Yaskawa INFORM job: pointsmerc2.JBI

'PP version: 0.3
/JOB
//NAME pointsmerc2
//POS
///NPOS 0,0,0,0,0,0
///TOOL 1
///POSTYPE ROBOT
///RECTAN
///RCONF 1,0,0,0,0,0,0,0,0,0,0,0,0,0,0,0,0,0,0,0,0,0,0,0
//INST
///DATE 2021/02/10 13:51
///COMM
///ATTR SC,RW,RJ
////FRAME USER 2
///GROUP1 RB1
///GROUP2 ST1
NOP
CALL JOB:DEBUT
'Part trajectory number: 0
CALL JOB:pointsmerc2TRJ0
'Part trajectory number: 1
CALL JOB:pointsmerc2TRJ1
'Part trajectory number: 2
CALL JOB:pointsmerc2TRJ2
CALL JOB:FIN
END
